Fanuc KAREL source: NC0045.compact.KL

PROGRAM NC0045
%STACKSIZE=65535
%PRIORITY=65535
%NOLOCKGROUP
ROUTINE R FROM NC0045
ROUTINE R
VAR
S1 : INTEGER
BEGIN
S1=1
IF (S1=1) THEN
SELECT S1 OF
CASE(1):
IF (S1=1) THEN
SELECT S1 OF
CASE(1):
IF (S1=1) THEN
S1=(S1 + 1)
ELSE
S1=(S1 + 2)
ENDIF
CASE(2):
S1=(S1 + 2)
ELSE:
S1=(S1 + 3)
ENDSELECT
ELSE
S1=(S1 + 2)
ENDIF
CASE(2):
S1=(S1 + 2)
ELSE:
S1=(S1 + 3)
ENDSELECT
ELSE
S1=(S1 + 2)
ENDIF
END R
BEGIN
R
END NC0045
